{attribute 'pack_mode' := '1'}
TYPE AxisStatus EXTENDS OutgoingMessage :
STRUCT
	axisIndex: DINT; (* 1 or 2. *)
	enabled: BOOL; (* Axis enabled? *)
	moving: BOOL;  (* Axis moving? *)
	homed: BOOL;   (* Axis has been homed? *)
	atLowLimit: BOOL; (* Axis at low limit switch? *)
	atHighLimit: BOOL; (* Axis at high limit switch? *)
	errorCode: DINT;
	position: LREAL;
END_STRUCT
END_TYPE

(* stored: Version 1.1.0.1, ProductVersion 3.1.4022.12
   DUT AxisStatus: Id {cf26e3e0-fe63-4d45-ac51-0519a8ae0daa} *)
